{attribute addProperty BoxType "EP1809-0042-0018"}
{attribute addProperty Id "InputAT %I*BOOL81"}
{attribute addProperty CRC "3836671390"}
{attribute addProperty SizeInBites "8"}
{attribute addProperty SizeInBytes "1"}
TYPE DI_X07_Pin_E4AEF59E :
STRUCT
	{attribute addProperty Name "Input"}
	Input AT %I* : BOOL;
END_STRUCT
END_TYPE

(* stored: Version 1.2.0.0, ProductVersion 3.1.4024.9
   DUT DI_X07_Pin_E4AEF59E: Id {48b7a6a3-a4cf-4601-96df-001535c54361} *)
